PROGRAM JIG_TAKER
VAR
END_VAR

END_PROGRAM

(* stored: Version 1.1.0.1, ProductVersion 3.1.4022.18
   POU JIG_TAKER: Id {56c7505f-2c83-448f-9292-c4eafd49cefb}, SpecialFunc None *)
